# B&R Automation Studio project Sim_Eksamen_Test11
Automation Studio 4.7.2.98

## Logical view

### Global.var
```iecst
VAR
	GoBtn : BOOL;
END_VAR
```

### Program Logical/Feed_Conv

#### Variables.var
```iecst
VAR
	TON_Timer : TON;
	doFeederMid : BOOL;
	doFeederLeft : BOOL;
	doFeederRight : BOOL;
	doConvMainStart : BOOL;
	FeedCount : USINT;
END_VAR
```

#### Main.st
```iecst
PROGRAM _INIT
	// Feeder timer initialization
	TON_Timer.PT := T#2s;

END_PROGRAM

PROGRAM _CYCLIC

	IF GoBtn THEN
		doConvMainStart := TRUE;
		TON_Timer.IN := TRUE;

		// Johans Feeder roundtable.
		IF FeedCount = 0 AND TON_Timer.Q THEN
			doFeederLeft := TRUE;
			doFeederRight := FALSE;
			FeedCount := 1;
			TON_Timer.IN := FALSE;
		ELSIF FeedCount = 1 AND TON_Timer.Q THEN
			doFeederMid := TRUE;
			doFeederLeft := FALSE;
			FeedCount := 2;
			TON_Timer.IN := FALSE;
		ELSIF FeedCount = 2 AND TON_Timer.Q THEN
			doFeederRight := TRUE;
			doFeederMid := FALSE;
			TON_Timer.IN := FALSE;
			FeedCount := 0;
		END_IF;

	ELSE
		// Reset all.
		doConvMainStart := FALSE;
		doFeederLeft := FALSE;
		doFeederMid := FALSE;
		doFeederRight := FALSE;
		TON_Timer.IN := FALSE;
	END_IF;

	// Functionblock Calls
	TON_Timer();
END_PROGRAM

PROGRAM _EXIT
	(* Insert code here *)

END_PROGRAM
```

### Program Logical/Sorter

#### Variables.var
```iecst
VAR
	doSorterPick : BOOL;
	diWeightScale : WORD;
	R_TRIG_RightPos : R_TRIG;
	R_TRIG_PickInitiated : R_TRIG;
	TON_DelayTimer : TON;
	sorterRobot : RobotArm;
	bigBoxDetected : BOOL;
END_VAR
```

#### Main.st
```iecst
PROGRAM _INIT
	// Timer initialization
	TON_DelayTimer.PT := T#1s;
END_PROGRAM

PROGRAM _CYCLIC
	R_TRIG_RightPos.CLK := bigBoxDetected;
	R_TRIG_PickInitiated.CLK := sorterRobot.Delivering;
	// Detecting bigBox
	IF diWeightScale > 300 THEN
		bigBoxDetected := TRUE;
	ELSE
		bigBoxDetected := FALSE;
	END_IF;

	IF GoBtn THEN

		// Weight gets activated.
		IF R_TRIG_RightPos.Q  THEN
			// If it's notv right, then we pick
			TON_DelayTimer.IN := TRUE;
		END_IF;

		// Delay timer for activating Sorter
		IF TON_DelayTimer.Q THEN
			TON_DelayTimer.IN := FALSE;
			doSorterPick := TRUE;
		END_IF;

		// Delay timer for switching input off. (Might be error if Blocks are too close to one another)
		IF R_TRIG_PickInitiated.Q THEN
			doSorterPick := FALSE;
		END_IF;

	ELSE
		// Reset all.
		TON_DelayTimer.IN := FALSE;
		doSorterPick := FALSE;

	END_IF;

	// Functionblock Calls
	TON_DelayTimer();
	R_TRIG_PickInitiated();
	R_TRIG_RightPos();
END_PROGRAM

PROGRAM _EXIT
	(* Insert code here *)

END_PROGRAM
```

### Program Logical/Stacker

#### Variables.var
```iecst
VAR
	doStackerPick : BOOL;
	diStackDone : BOOL;
	R_TRIG_diGoBtn : R_TRIG;
	R_TRIG_StackerCount : R_TRIG;
	R_TRIG_StackDone : R_TRIG;
	doConvSideStart : BOOL;
	diPlateBoxBlocked : BOOL;
	F_TRIG_StackDone : F_TRIG;
	F_TRIG_BoxBlocked : F_TRIG;
	doStackerInputBelt : BOOL;
	diStackerInputSensor : BOOL;
	stackCount : USINT;
	doResetStackers : BOOL;
	diGoBtn : BOOL;
END_VAR
```

#### Main.st
```iecst
PROGRAM _INIT
		(* Insert code here *)

END_PROGRAM

PROGRAM _CYCLIC
	R_TRIG_StackDone.CLK := diStackDone;
	R_TRIG_diGoBtn.CLK := diGoBtn;
	F_TRIG_BoxBlocked.CLK := diPlateBoxBlocked;
	R_TRIG_StackerCount.CLK := diStackerInputSensor;
	F_TRIG_StackDone.CLK := diStackDone;
	GoBtn := diGoBtn;

	IF GoBtn THEN
		// Stop belt when box is exactly in place.
		doStackerInputBelt := NOT diStackerInputSensor;

		// Increase count on rising edge.
		IF R_TRIG_StackerCount.Q THEN
			stackCount := stackCount +1;
		END_IF;

		// Initiate plate serving in start of program.
		IF R_TRIG_diGoBtn.Q THEN
			doConvSideStart := TRUE;
		END_IF;

		// Move output belt when the stack is stacked,
		IF R_TRIG_StackDone.Q THEN
			doConvSideStart := TRUE;
		END_IF;
		// and stop it again.
		IF F_TRIG_BoxBlocked.Q THEN
			doConvSideStart := FALSE;
			// Reset count according to wether a block is ready for pickup or not.
			IF diStackerInputSensor THEN
				stackCount := 1;
			ELSE
				stackCount := 0;
			END_IF;

			// Reset for stackers
			IF diStackDone THEN
				doResetStackers := TRUE;
			END_IF;
		END_IF;

		// Activate stackers
		doStackerPick := diStackerInputSensor AND
						 NOT (stackCount > 8) AND
						 NOT doConvSideStart AND
						 NOT diStackDone;

		// Reset stacker Reset
		IF F_TRIG_StackDone.Q THEN
			doResetStackers := FALSE;
		END_IF;
	ELSE
		// Reset all.
		doStackerPick := FALSE;
		doConvSideStart := FALSE;
		doStackerInputBelt := FALSE;
		stackCount := 0;
	END_IF;

	// Functionblock Calls
	R_TRIG_StackDone();
	R_TRIG_diGoBtn();
	F_TRIG_BoxBlocked();
	R_TRIG_StackerCount();
	F_TRIG_StackDone();
END_PROGRAM

PROGRAM _EXIT
	(* Insert code here *)

END_PROGRAM
```
